// TIA Portal V20 export
DATA_BLOCK "InstProductionDataMove"   // DB40120
// stored: InstanceOfName Count, InstanceOfType FB
"Count"
   // VAR
   //    statPulse { ExternalAccessible := 'False'; ExternalVisible := 'False'; ExternalWritable := 'False'} : Array[0..299] of Bool;
   // END_VAR
BEGIN
END_DATA_BLOCK
